// Mitsubishi GX Works2 project: 240416_주기동작회로   PLC: Q03UDV

PROGRAM MAIN
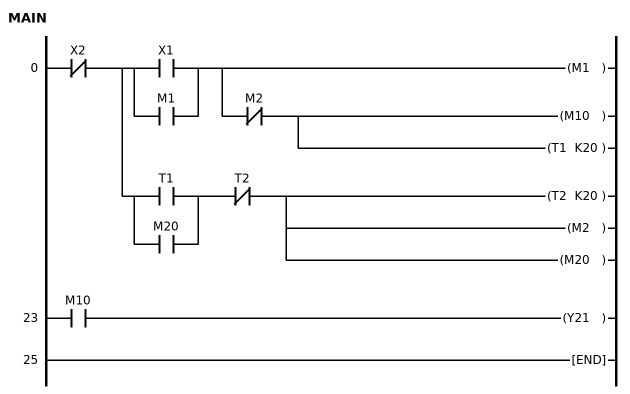
0     LDI     X2
      MPS
      LD      X1
      OR      M1
      ANB
      OUT     M1
      ANI     M2
      OUT     M10
      OUT     T1 K20
      MPP
      LD      T1
      OR      M20
      ANB
      ANI     T2
      OUT     T2 K20
      OUT     M2
      OUT     M20
23    LD      M10
      OUT     Y21
25    END
END_PROGRAM

PROGRAM OUTPUT
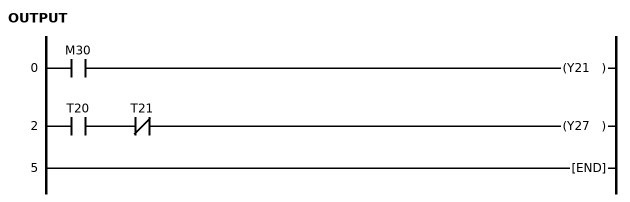
0     LD      M30
      OUT     Y21
2     LD      T20
      ANI     T21
      OUT     Y27
5     END
END_PROGRAM

PROGRAM OYTPUT1
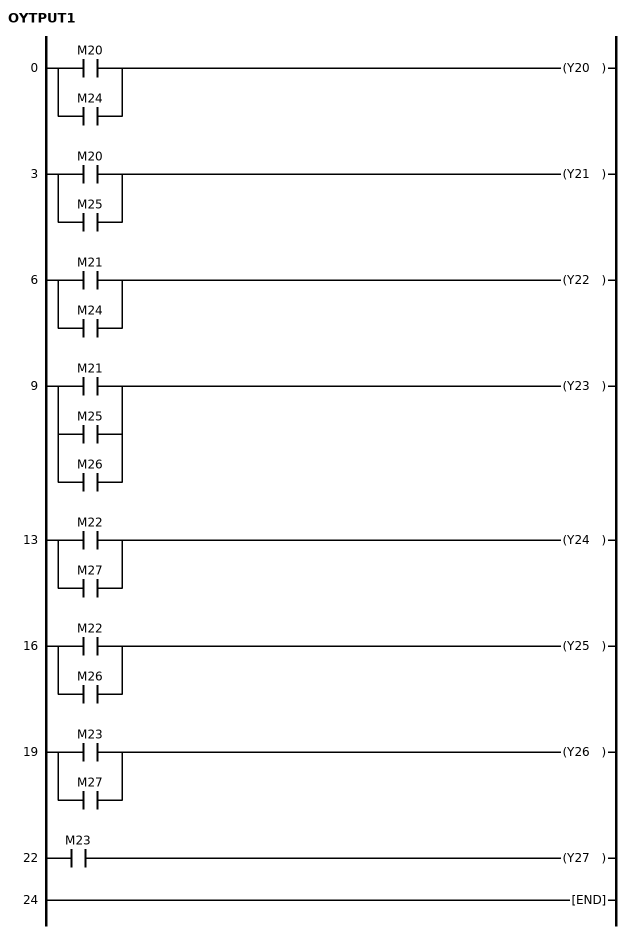
0     LD      M20
      OR      M24
      OUT     Y20
3     LD      M20
      OR      M25
      OUT     Y21
6     LD      M21
      OR      M24
      OUT     Y22
9     LD      M21
      OR      M25
      OR      M26
      OUT     Y23
13    LD      M22
      OR      M27
      OUT     Y24
16    LD      M22
      OR      M26
      OUT     Y25
19    LD      M23
      OR      M27
      OUT     Y26
22    LD      M23
      OUT     Y27
24    END
END_PROGRAM

PROGRAM OUTPUT1
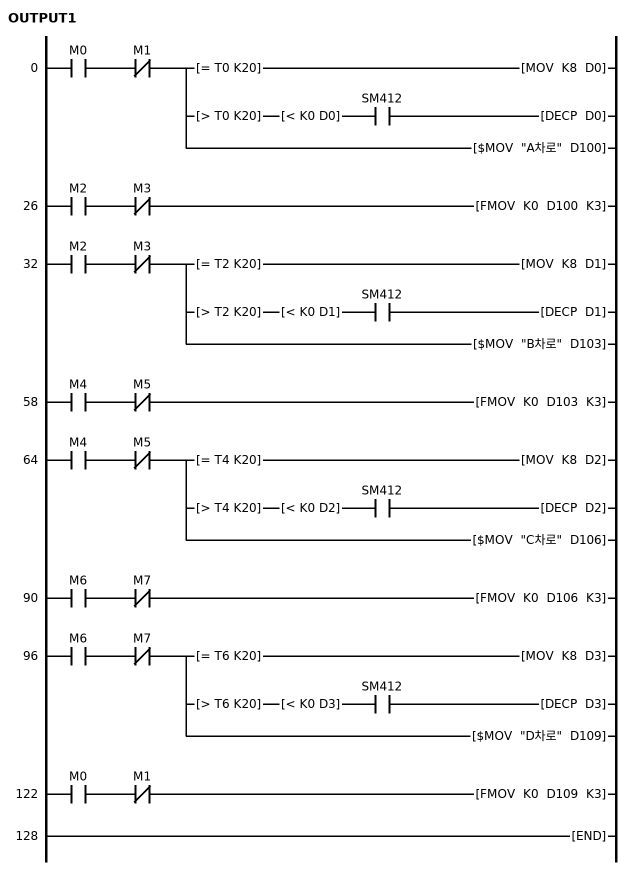
0     LD      M0
      ANI     M1
      MPS
      AND=    T0 K20
      MOV     K8 D0
      MRD
      AND>    T0 K20
      AND<    K0 D0
      AND     SM412
      DECP    D0
      MPP
      $MOV    "A차로" D100
26    LD      M2
      ANI     M3
      FMOV    K0 D100 K3
32    LD      M2
      ANI     M3
      MPS
      AND=    T2 K20
      MOV     K8 D1
      MRD
      AND>    T2 K20
      AND<    K0 D1
      AND     SM412
      DECP    D1
      MPP
      $MOV    "B차로" D103
58    LD      M4
      ANI     M5
      FMOV    K0 D103 K3
64    LD      M4
      ANI     M5
      MPS
      AND=    T4 K20
      MOV     K8 D2
      MRD
      AND>    T4 K20
      AND<    K0 D2
      AND     SM412
      DECP    D2
      MPP
      $MOV    "C차로" D106
90    LD      M6
      ANI     M7
      FMOV    K0 D106 K3
96    LD      M6
      ANI     M7
      MPS
      AND=    T6 K20
      MOV     K8 D3
      MRD
      AND>    T6 K20
      AND<    K0 D3
      AND     SM412
      DECP    D3
      MPP
      $MOV    "D차로" D109
122   LD      M0
      ANI     M1
      FMOV    K0 D109 K3
128   END
END_PROGRAM

PROGRAM OUTPUT2
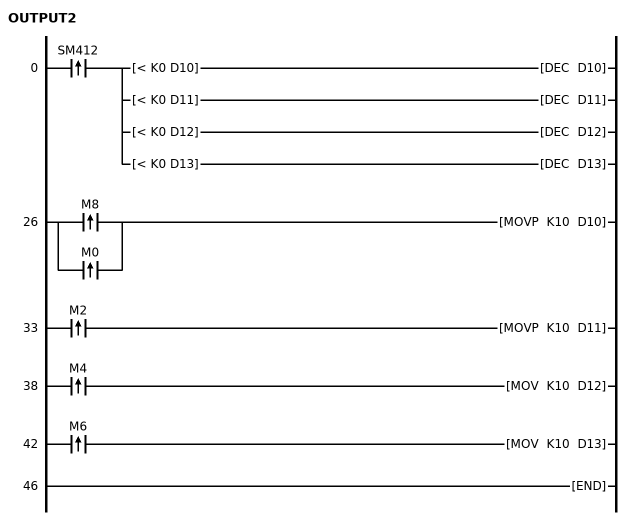
0     LDP     SM412
      MPS
      AND<    K0 D10
      DEC     D10
      MRD
      AND<    K0 D11
      DEC     D11
      MRD
      AND<    K0 D12
      DEC     D12
      MPP
      AND<    K0 D13
      DEC     D13
26    LDP     M8
      ORP     M0
      MOVP    K10 D10
33    LDP     M2
      MOVP    K10 D11
38    LDP     M4
      MOV     K10 D12
42    LDP     M6
      MOV     K10 D13
46    END
END_PROGRAM

PROGRAM MAIN1
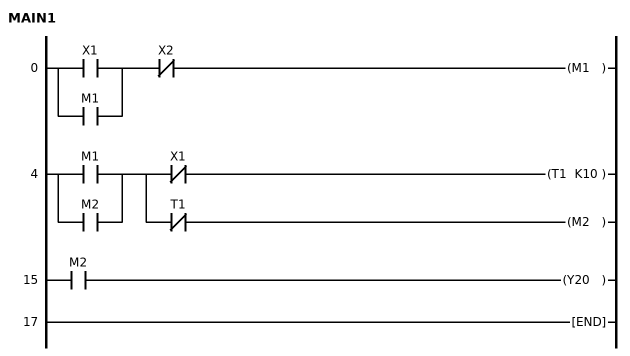
0     LD      X1
      OR      M1
      ANI     X2
      OUT     M1
4     LD      M1
      OR      M2
      MPS
      ANI     X1
      OUT     T1 K10
      MPP
      ANI     T1
      OUT     M2
15    LD      M2
      OUT     Y20
17    END
END_PROGRAM
